# EPICS autosave request: iocBoot/iocrunControl/auto_positions.req
file runControl_settings.req P=$(P)
$(P)CAM_PIXEL_SIZE_X
$(P)SAMPLE_ID
$(P)SINE_PHOSPHOR
$(P)SS_G0_DIST
$(P)SS_G1_DIST
$(P)SS_SAMPLE_DIST
$(P)SS_G2_DIST
$(P)SS_DET_DIST
$(P)PHOSPHOR_TYPE
$(P)INVESTIGATOR
$(P)METADATA_1
